// TIA Portal project "Alarms" (V15.1)

(* hardware
DEVICE "S71500/ET200MP station_1"  S7-1500 station
   slot 0: "Rail_0"  Rack  6ES7 590-1***0-0AA0
   slot 0: "PM 190W 120/230VAC"  PM 190W 120/230VAC  6EP1333-4BA00
   slot 1: "PLC_1"  CPU 1516-3 PN/DP  6ES7 516-3AN01-0AB0  V2.6
      slot 3: "CPU display_1"  6ES7591-1BA00-0AA0
   slot 2: "DQ 32x24VDC/0.5A HF_1"  DQ 32x24VDC/0.5A HF  6ES7 522-1BL01-0AB0  V1.1
   slot 3: "DI 32x24VDC HF_1"  DI 32x24VDC HF  6ES7 521-1BL00-0AB0  V2.1
   slot 4: "AQ 4xU/I ST_1"  AQ 4xU/I ST  6ES7 532-5HD00-0AB0  V2.2
   slot 5: "AI 8xU/I/RTD/TC ST_1"  AI 8xU/I/RTD/TC ST  6ES7 531-7KF00-0AB0  V2.2
DEVICE "HMI_1"  TP700 Comfort
   slot 0: "HMI_1"  TP700 Comfort  6AV2 124-0GC01-0AX0  15.1.0.0
   slot 1: "HMI_RT_1"  TP700 Comfort  6AV2 124-0GC01-0AX0  15.1.0.0
   slot 5: "HMI_1.IE_CP_1"  PROFINET Interface  15.0.1.0
      slot 1: "PROFINET Interface_1"  PROFINET Interface
         slot 1: "Port_1"  Port
         slot 2: "Port_2"  Port
   slot 7: "HMI_1.MPI/DP_CP_1"  MPI/DP Interface  15.0.1.0
*)

// ===== PLC "PLC_1"  CPU 1516-3 PN/DP =====

VAR_GLOBAL   // PLC tag table "Default tag table"
   "Clock_Byte" AT %MB0 : Byte;
   "Clock_10Hz" AT %M0.0 : Bool;
   "Clock_5Hz" AT %M0.1 : Bool;
   "Clock_2.5Hz" AT %M0.2 : Bool;
   "Clock_2Hz" AT %M0.3 : Bool;
   "Clock_1.25Hz" AT %M0.4 : Bool;
   "Clock_1Hz" AT %M0.5 : Bool;
   "Clock_0.625Hz" AT %M0.6 : Bool;
   "Clock_0.5Hz" AT %M0.7 : Bool;
   "System_Byte" AT %MB1 : Byte;
   "FirstScan" AT %M1.0 : Bool;
   "DiagStatusUpdate" AT %M1.1 : Bool;
   "AlwaysTRUE" AT %M1.2 : Bool;
   "AlwaysFALSE" AT %M1.3 : Bool;
   "System_Byte(1)" AT %MB1 : Byte;
   "System_Byte(2)" AT %MB1 : Byte;
END_VAR

VAR_GLOBAL   // PLC tag table "Full_Tag_Table"
   "Panel Emergency Stop" AT %I2.7 : Bool;
   "Start switch" AT %I0.2 : Bool;
   "Stop switch" AT %I0.3 : Bool;
   "Sort area IR" AT %I0.4 : Bool;
   "Sort Area Inductive" AT %I0.5 : Bool;
   "Sort Solenoid Sensor" AT %I0.6 : Bool;
   "Assembly Chute IR" AT %I0.7 : Bool;
   "Assembly Area Through Beam" AT %I1.1 : Bool;
   "Assembly Area Capacitor" AT %I1.2 : Bool;
   "Assembly Area Inductive" AT %I1.3 : Bool;
   "Reject Area IR" AT %I1.4 : Bool;
   "Reject Solenoid Sensor" AT %I1.5 : Bool;
   "Oven Through Beam" AT %I1.6 : Bool;
   "Loading Area Inductive" AT %I1.7 : Bool;
   "Chain Conveyor" AT %Q0.0 : Bool;
   "Sort Solenoid" AT %Q0.1 : Bool;
   "Reject Solenoid" AT %Q0.2 : Bool;
   "Rotary Solenoid" AT %Q0.3 : Bool;
   "Belt Conveyor Direction" AT %Q0.4 : Bool;
   "System Run_Green Lamp" AT %Q3.0 : Bool;
   "Sysyem Stop_Red Lamp" AT %Q3.2 : Bool;
   "Emergency stop" AT %I1.0 : Bool;
   "Ring Queue counter Full" AT %M4.0 : Bool;
   "Sort Solenoid error" AT %M4.3 : Bool;
   "Counter value" AT %MW0 : Int;
   "Reject Solenoid Error" AT %M4.7 : Bool;
   "HMI_Start" AT %M4.1 : Bool;
   "HMI_Stop" AT %M4.2 : Bool;
   "Counter Reset" AT %M4.4 : Bool;
   "Assembly Complete" AT %M4.5 : Bool;
   "Reset" AT %M4.6 : Bool;
   "HMI_Emergency_Stop" AT %M5.0 : Bool;
   "Ring Counter Value" AT %MW2 : Int;
   "Peg Counter Value" AT %MW6 : Int;
   "Assembly Counter Value" AT %MW8 : Int;
   "Connection_Successful" AT %M5.1 : Bool;
   "Connection_Disconnected" AT %M5.2 : Bool;
   "HMI_AssemDone" AT %M5.3 : Bool;
   "HMI_ConReset" AT %M5.4 : Bool;
   "HMI_SS_Alarm" AT %MW5 : Int;
   "Oven Temperature" AT %IW4 : Int;
   "Temperature control" AT %QW4 : Int;
   "Bipolar_SCALE" AT %M2000.0 : Bool;
   "Bipolar_UNSCALE" AT %M2000.1 : Bool;
   "Actual Retain Value" AT %MW100 : Word;
   "UNSCALE retain value" AT %MW15 : Word;
   "Real Temperature" AT %MD300 : Real;
   "Control value" AT %MW13 : Int;
   "ON/OFF Temperature" AT %MD9 : Real;
   "Temperature set point" AT %MD24 : Real;
   "ON/OFF Temperature set point" AT %MD20 : Real;
   "Save_Energy" AT %M28.0 : Bool;
   "Reset2" AT %M28.2 : Bool;
   "Em_Alarm" AT %M20.0 : Bool;
   "Alarm_Tag" AT %MW20 : Int;
   "PaEm_Alarm" AT %M20.1 : Bool;
   "SortSole_Alarm" AT %M20.2 : Bool;
   "RejectSole_Alarm" AT %M20.3 : Bool;
   "Count_Alarm" AT %M20.4 : Bool;
   "HMIReset" AT %M6.0 : Bool;
END_VAR

DATA_BLOCK "Automatic_Conveyor_DB"   // DB1
{ S7_Optimized_Access := 'TRUE' }
VERSION : 0.1
// stored: InstanceOfName Automatic_Conveyor
"Automatic_Conveyor"
BEGIN
END_DATA_BLOCK

DATA_BLOCK "Sort Solenoid Active_DB"   // DB2
{ S7_Optimized_Access := 'TRUE' }
VERSION : 0.1
// stored: InstanceOfName Sort Solenoid Active
"Sort Solenoid Active"
BEGIN
END_DATA_BLOCK

DATA_BLOCK "Solenoids Error_DB"   // DB3
{ S7_Optimized_Access := 'TRUE' }
VERSION : 0.1
// stored: InstanceOfName Solenoids Error
"Solenoids Error"
BEGIN
END_DATA_BLOCK

DATA_BLOCK "Rotary Solenoid Active_DB"   // DB4
{ S7_Optimized_Access := 'TRUE' }
VERSION : 0.1
// stored: InstanceOfName Rotary Solenoid Active
"Rotary Solenoid Active"
BEGIN
END_DATA_BLOCK

DATA_BLOCK "Counting_DB"   // DB5
{ S7_Optimized_Access := 'TRUE' }
VERSION : 0.1
// stored: InstanceOfName Counting
"Counting"
BEGIN
END_DATA_BLOCK

DATA_BLOCK "Solenoids Error_DB_1"   // DB6
{ S7_Optimized_Access := 'TRUE' }
VERSION : 0.1
// stored: InstanceOfName Solenoids Error
"Solenoids Error"
BEGIN
END_DATA_BLOCK

DATA_BLOCK "Component Queue Handling_DB"   // DB7
{ S7_Optimized_Access := 'TRUE' }
VERSION : 0.1
// stored: InstanceOfName Component Queue Handling
"Component Queue Handling"
BEGIN
END_DATA_BLOCK

DATA_BLOCK "Datablock"   // DB12
{ S7_Optimized_Access := 'TRUE' }
VERSION : 0.1
   VAR
      Sending_Data : Array[0..12] of Byte;
      Received_Data : Array[0..10] of Char;
      Send_Comm : Array[0..15] of Char;
   END_VAR
BEGIN
   Sending_Data[0] := 'A';
   Sending_Data[1] := 's';
   Sending_Data[2] := 's';
   Sending_Data[3] := 'e';
   Sending_Data[4] := 'm';
   Sending_Data[5] := 'b';
   Sending_Data[6] := 'l';
   Sending_Data[7] := 'y';
   Sending_Data[8] := ' ';
   Sending_Data[9] := 'D';
   Sending_Data[10] := 'o';
   Sending_Data[11] := 'n';
   Sending_Data[12] := 'e';
   Send_Comm[2] := 'o';
   Send_Comm[1] := 'r';
   Send_Comm[0] := 'P';
   Send_Comm[3] := 'c';
   Send_Comm[4] := 'e';
   Send_Comm[5] := 's';
   Send_Comm[6] := 's';
   Send_Comm[7] := ' ';
   Send_Comm[8] := 'S';
   Send_Comm[9] := 't';
   Send_Comm[10] := 'a';
   Send_Comm[11] := 'r';
   Send_Comm[12] := 't';
   Send_Comm[13] := 'e';
   Send_Comm[14] := 'd';
   Send_Comm[15] := '!';
END_DATA_BLOCK

DATA_BLOCK "TCP/IP Connection_DB"   // DB14
{ S7_Optimized_Access := 'TRUE' }
VERSION : 0.1
// stored: InstanceOfName TCP/IP Connection
"TCP/IP Connection"
BEGIN
END_DATA_BLOCK

DATA_BLOCK "Energy Saving_DB"   // DB17
{ S7_Optimized_Access := 'TRUE' }
VERSION : 0.1
// stored: InstanceOfName Energy Saving
"Energy Saving"
BEGIN
END_DATA_BLOCK

DATA_BLOCK "Alarm_DB"   // DB18
{ S7_Optimized_Access := 'TRUE' }
VERSION : 0.1
// stored: InstanceOfName Alarm
"Alarm"
BEGIN
END_DATA_BLOCK

// folder: System blocks/Program resources

DATA_BLOCK "PLC_1_Connection_DB"   // DB13
{ S7_Optimized_Access := 'TRUE' }
AUTHOR : SIMATIC
FAMILY : MC7Plus
NAME : TC_IP_v4
VERSION : 1.0
// stored: InstanceOfName TCON_IP_v4
"TCON_IP_v4"
BEGIN
   ID := 1;
   InterfaceId := 64;
   LocalPort := 2000;
   RemotePort := 10999;
   ActiveEstablished := true;
   RemoteAddress.ADDR[1] := 192;
   RemoteAddress.ADDR[2] := 168;
   RemoteAddress.ADDR[4] := 3;
END_DATA_BLOCK

// folder: (top level)

FUNCTION_BLOCK "Automatic_Conveyor"   // FB1, LAD
TITLE = Conveyors Automatic
{ S7_Optimized_Access := 'TRUE' }
VERSION : 0.1
   VAR_INPUT
      "Start Switch" : Bool;
      "Stop Switch" : Bool;
      "Emergency Stop" : Bool;
      "Panel Emergency Stop" : Bool;
      "Sort Solenoid Error" : Bool;
      "Reject Solenoid Error" : Bool;
      Reset : Bool;
      "Assembly Done" : Bool;
      H_Start : Bool;
      H_Stop : Bool;
      H_Emer_Stop : Bool;
      Save : Bool;
   END_VAR
   VAR_OUTPUT
      "System Enable_OK" : Bool;
      "System Enable_not_OK" : Bool;
      "Chain Conveyor" : Bool;
      "Belt Conveyor" : Bool;
   END_VAR
   VAR_IN_OUT
      Reset2 : Bool;
   END_VAR
   VAR
      Memory_Automatic_Start_Stop : Bool;
      Temp : Bool;
      SR_Temp : Bool;
      IEC_Timer_0_Instance_1 : TON_TIME;
      IEC_Timer_0_Instance_3 : TON_TIME;
   END_VAR
BEGIN

REGION Network 1: System Enable_OK and Conveyors run
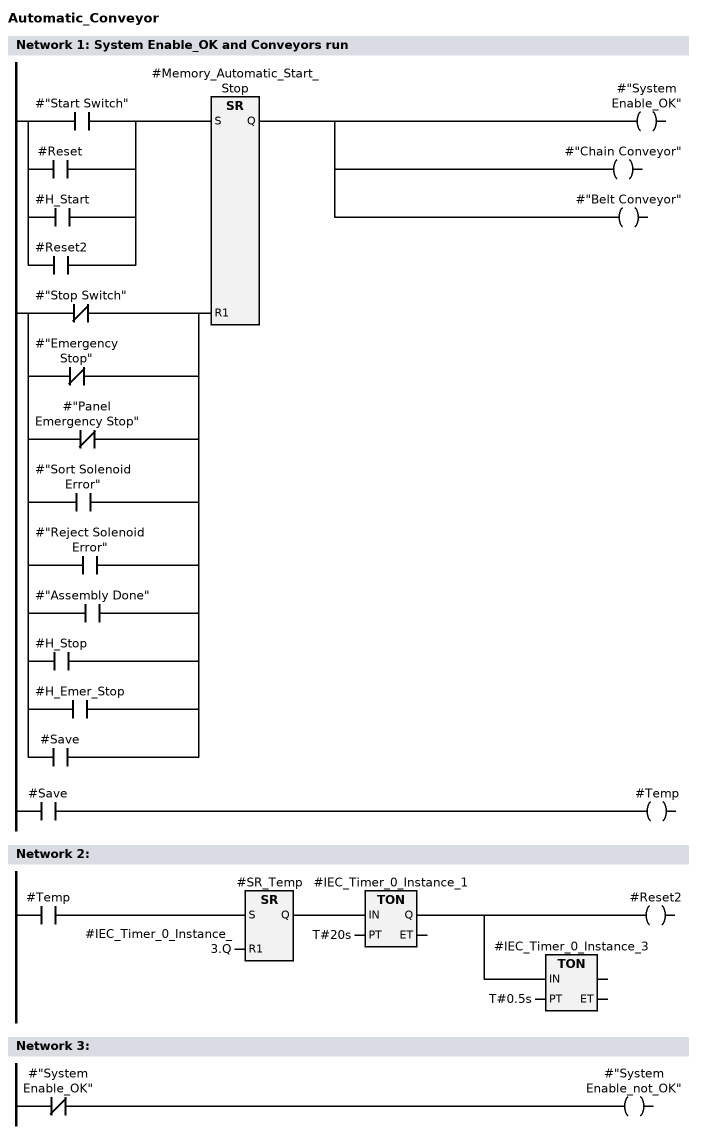
   RUNG wire#powerrail
      Contact( #"Start Switch" )
      wire#w1
      S_SR(operand := #Memory_Automatic_Start_Stop, r1 := wire#w2)
      wire#w3
      Coil( #"System Enable_OK" )
   END_RUNG
   RUNG wire#powerrail
      Contact( #Reset )
   END_RUNG wire#w1
   RUNG wire#powerrail
      Contact( #H_Start )
   END_RUNG wire#w1
   RUNG wire#powerrail
      Contact( #Reset2 )
   END_RUNG wire#w1
   RUNG wire#powerrail
      I_Contact( #"Stop Switch" )
   END_RUNG wire#w2
   RUNG wire#powerrail
      I_Contact( #"Emergency Stop" )
   END_RUNG wire#w2
   RUNG wire#powerrail
      I_Contact( #"Panel Emergency Stop" )
   END_RUNG wire#w2
   RUNG wire#powerrail
      Contact( #"Sort Solenoid Error" )
   END_RUNG wire#w2
   RUNG wire#powerrail
      Contact( #"Reject Solenoid Error" )
   END_RUNG wire#w2
   RUNG wire#powerrail
      Contact( #"Assembly Done" )
   END_RUNG wire#w2
   RUNG wire#powerrail
      Contact( #H_Stop )
   END_RUNG wire#w2
   RUNG wire#powerrail
      Contact( #H_Emer_Stop )
   END_RUNG wire#w2
   RUNG wire#powerrail
      Contact( #Save )
   END_RUNG wire#w2
   RUNG wire#w3
      Coil( #"Chain Conveyor" )
   END_RUNG
   RUNG wire#w3
      Coil( #"Belt Conveyor" )
   END_RUNG
   RUNG wire#powerrail
      Contact( #Save )
      Coil( #Temp )
   END_RUNG
   // the same network as SCL:
   IF #"Start Switch" OR #Reset OR #H_Start OR #Reset2 THEN
       #Memory_Automatic_Start_Stop := TRUE;   // SR flip-flop
   END_IF;
   IF NOT #"Stop Switch" OR NOT #"Emergency Stop" OR NOT #"Panel Emergency Stop" OR #"Sort Solenoid Error" OR #"Reject Solenoid Error" OR #"Assembly Done" OR #H_Stop OR #H_Emer_Stop OR #Save THEN
       #Memory_Automatic_Start_Stop := FALSE;
   END_IF;
   #"System Enable_OK" := #Memory_Automatic_Start_Stop;
   #"Chain Conveyor" := #Memory_Automatic_Start_Stop;
   #"Belt Conveyor" := #Memory_Automatic_Start_Stop;
   #Temp := #Save;
END_REGION

REGION Network 2
   IF #Temp THEN
       #SR_Temp := TRUE;   // SR flip-flop
   END_IF;
   IF #IEC_Timer_0_Instance_3.Q THEN #SR_Temp := FALSE; END_IF;
   #IEC_Timer_0_Instance_1(IN := #SR_Temp, PT := T#20s);   // TON
   #Reset2 := #IEC_Timer_0_Instance_1.Q;
   #IEC_Timer_0_Instance_3(IN := #IEC_Timer_0_Instance_1.Q, PT := T#0.5s);   // TON
END_REGION

REGION Network 3
   RUNG wire#powerrail
      I_Contact( #"System Enable_OK" )
      Coil( #"System Enable_not_OK" )
   END_RUNG
   // the same network as SCL:
   #"System Enable_not_OK" := NOT #"System Enable_OK";
END_REGION
END_FUNCTION_BLOCK

FUNCTION_BLOCK "Sort Solenoid Active"   // FB2, LAD
TITLE = Sort Solenoid Active
{ S7_Optimized_Access := 'TRUE' }
VERSION : 0.1
   VAR_INPUT
      "Sort Area IR" : Bool;
      "Sort Area Inductive" : Bool;
      "Ring Counter Full" : Bool;
   END_VAR
   VAR_OUTPUT
      "Sort Solenoid" : Bool;
   END_VAR
   VAR
      "Component Pass Delay" : Bool;
      "SR_Sort Solenoid on Timer" : Bool;
      "SR_Component Pass Delay" : Bool;
      IEC_Timer_0_Instance : TON_TIME;
      IEC_Timer_0_Instance_2 : TON_TIME;
   END_VAR
BEGIN

REGION Network 1: Sort Solenoid Active if Plastic Ring Present
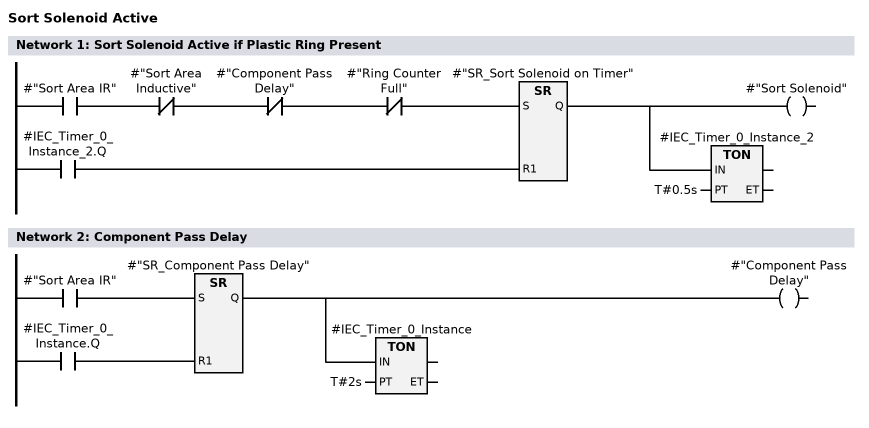
   IF #"Sort Area IR" AND NOT #"Sort Area Inductive" AND NOT #"Component Pass Delay" AND NOT #"Ring Counter Full" THEN
       #"SR_Sort Solenoid on Timer" := TRUE;   // SR flip-flop
   END_IF;
   IF #IEC_Timer_0_Instance_2.Q THEN #"SR_Sort Solenoid on Timer" := FALSE; END_IF;
   #"Sort Solenoid" := #"SR_Sort Solenoid on Timer";
   #IEC_Timer_0_Instance_2(IN := #"SR_Sort Solenoid on Timer", PT := T#0.5s);   // TON
END_REGION

REGION Network 2: Component Pass Delay
   IF #"Sort Area IR" THEN
       #"SR_Component Pass Delay" := TRUE;   // SR flip-flop
   END_IF;
   IF #IEC_Timer_0_Instance.Q THEN #"SR_Component Pass Delay" := FALSE; END_IF;
   #"Component Pass Delay" := #"SR_Component Pass Delay";
   #IEC_Timer_0_Instance(IN := #"SR_Component Pass Delay", PT := T#2s);   // TON
END_REGION
END_FUNCTION_BLOCK

FUNCTION_BLOCK "Solenoids Error"   // FB3, LAD
TITLE = Solenoid Error - Closed Loop Control
{ S7_Optimized_Access := 'TRUE' }
VERSION : 0.1
   VAR_INPUT
      "Solenoid on" : Bool;
      "Solenoid sensor" : Bool;
   END_VAR
   VAR_OUTPUT
      "Solenoid Error" : Bool;
   END_VAR
   VAR
      "Hold off delay" : Bool;
      IEC_Timer_0_Instance : TON_TIME;
   END_VAR
BEGIN

REGION Network 1: Solenoid Error
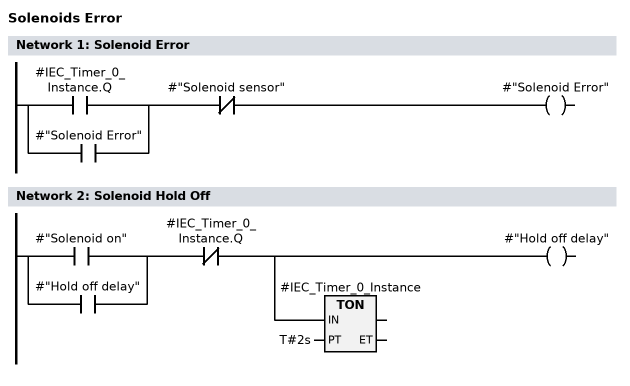
   RUNG wire#powerrail
      Contact( #IEC_Timer_0_Instance.Q )
      wire#w1
      I_Contact( #"Solenoid sensor" )
      Coil( #"Solenoid Error" )
   END_RUNG
   RUNG wire#powerrail
      Contact( #"Solenoid Error" )
   END_RUNG wire#w1
   // the same network as SCL:
   #"Solenoid Error" := (#IEC_Timer_0_Instance.Q OR #"Solenoid Error") AND NOT #"Solenoid sensor";
END_REGION

REGION Network 2: Solenoid Hold Off
   #"Hold off delay" := (#"Solenoid on" OR #"Hold off delay") AND NOT #IEC_Timer_0_Instance.Q;
   #IEC_Timer_0_Instance(IN := #"Hold off delay", PT := T#2s);   // TON
END_REGION
END_FUNCTION_BLOCK

FUNCTION_BLOCK "Counting"   // FB4, LAD
TITLE = Counting
{ S7_Optimized_Access := 'TRUE' }
VERSION : 0.1
// Incremental and Decremental counting
   VAR_INPUT
      "Sort Solenoid" : Bool;
      "Rotary Solenoid" : Bool;
      "Counter Reset" : Bool;
      "Sort Area Inductive" : Bool;
      "Sort Area IR" : Bool;
      "Assembly Complete" : Bool;
   END_VAR
   VAR_OUTPUT
      "Ring Queue counter full" : Bool;
      "Counter Value" : Int;
      "Ring CounterValue" : Int;
      "Peg CounterValue" : Int;
      "AssemblyCom CounterValue" : Int;
   END_VAR
   VAR RETAIN
      IEC_Counter_0_Instance : CTUD_INT;
      IEC_Counter_0_Instance_1 : CTU_INT;
      IEC_Counter_0_Instance_2 : CTU_INT;
      IEC_Counter_0_Instance_3 : CTU_INT;
   END_VAR
   VAR
      "Peg Count" : Bool;
      IEC_Timer_0_Instance : TOF_TIME;
   END_VAR
BEGIN

REGION Network 1: Counting
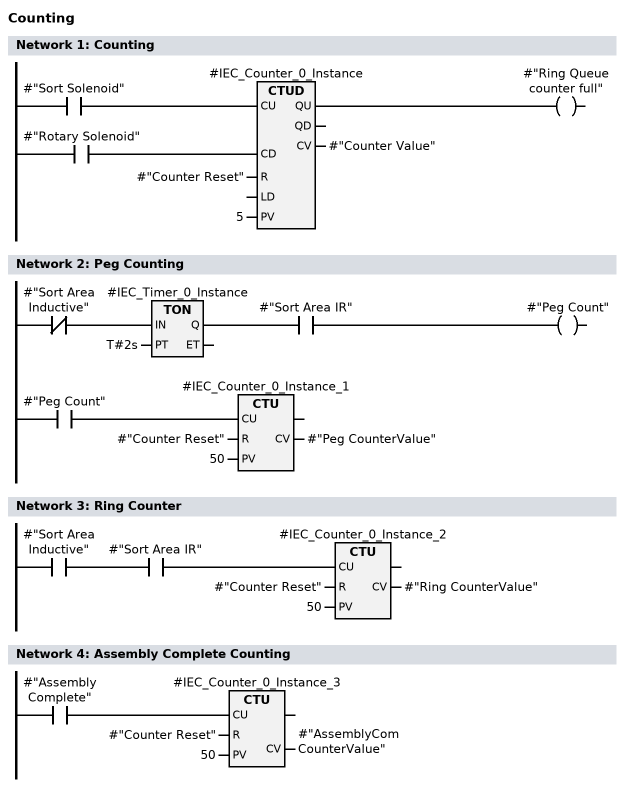
   #IEC_Counter_0_Instance(CU := #"Sort Solenoid",   // CTUD
                           CD := #"Rotary Solenoid",
                           R := #"Counter Reset",
                           PV := 5,
                           CV => #"Counter Value");
   #"Ring Queue counter full" := #IEC_Counter_0_Instance.QU;
END_REGION

REGION Network 2: Peg Counting
   #IEC_Timer_0_Instance(IN := NOT #"Sort Area Inductive", PT := T#2s);   // TON
   #"Peg Count" := #IEC_Timer_0_Instance.Q AND #"Sort Area IR";
   #IEC_Counter_0_Instance_1(CU := #"Peg Count", R := #"Counter Reset", PV := 50, CV => #"Peg CounterValue");   // CTU
END_REGION

REGION Network 3: Ring Counter
   #IEC_Counter_0_Instance_2(CU := #"Sort Area Inductive" AND #"Sort Area IR",   // CTU
                           R := #"Counter Reset",
                           PV := 50,
                           CV => #"Ring CounterValue");
END_REGION

REGION Network 4: Assembly Complete Counting
   #IEC_Counter_0_Instance_3(CU := #"Assembly Complete",   // CTU
                           R := #"Counter Reset",
                           PV := 50,
                           CV => #"AssemblyCom CounterValue");
END_REGION
END_FUNCTION_BLOCK

FUNCTION_BLOCK "Rotary Solenoid Active"   // FB5, LAD
TITLE = Rotary Solenoid Active
{ S7_Optimized_Access := 'TRUE' }
VERSION : 0.1
   VAR_INPUT
      "Rotary Area IR" : Bool;
   END_VAR
   VAR_OUTPUT
      "Rotary Solenoid" : Bool;
   END_VAR
   VAR
      "SR_Component Pass Delay" : Bool;
      "Component Pass Delay" : Bool;
      IEC_Timer_0_Instance : TON_TIME;
      IEC_Timer_0_Instance_2 : TON_TIME;
      "SR Rotary Solenoid on Timer" : Bool;
      IEC_Timer_0_Instance_1 : TON_TIME;
   END_VAR
BEGIN

REGION Network 1: Rotary Solenoid Activation
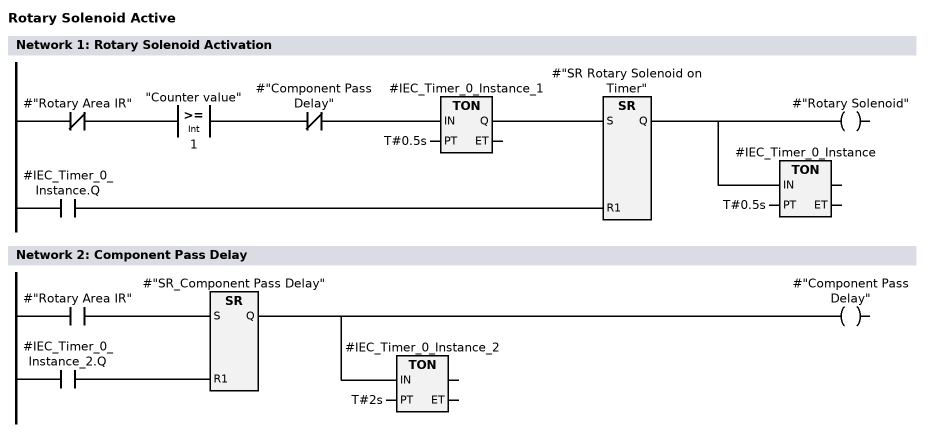
   #IEC_Timer_0_Instance_1(IN := NOT #"Rotary Area IR" AND ("Counter value" >= 1) AND NOT #"Component Pass Delay",   // TON
                           PT := T#0.5s);
   IF #IEC_Timer_0_Instance_1.Q THEN
       #"SR Rotary Solenoid on Timer" := TRUE;   // SR flip-flop
   END_IF;
   IF #IEC_Timer_0_Instance.Q THEN #"SR Rotary Solenoid on Timer" := FALSE; END_IF;
   #"Rotary Solenoid" := #"SR Rotary Solenoid on Timer";
   #IEC_Timer_0_Instance(IN := #"SR Rotary Solenoid on Timer", PT := T#0.5s);   // TON
END_REGION

REGION Network 2: Component Pass Delay
   IF #"Rotary Area IR" THEN
       #"SR_Component Pass Delay" := TRUE;   // SR flip-flop
   END_IF;
   IF #IEC_Timer_0_Instance_2.Q THEN #"SR_Component Pass Delay" := FALSE; END_IF;
   #"Component Pass Delay" := #"SR_Component Pass Delay";
   #IEC_Timer_0_Instance_2(IN := #"SR_Component Pass Delay", PT := T#2s);   // TON
END_REGION
END_FUNCTION_BLOCK

FUNCTION_BLOCK "Component Queue Handling"   // FB6, LAD
TITLE = Component Queue Handling
{ S7_Optimized_Access := 'TRUE' }
VERSION : 0.1
   VAR_INPUT
      "Start Switch" : Bool;
      "Assembly Area Capacitive" : Bool;
      "Assembly Area Inductive" : Bool;
      "Reject Area IR" : Bool;
      "Assembly Area Through Beam" : Bool;
   END_VAR
   VAR_OUTPUT
      "Reject Solenoid" : Bool;
      "Assembly Done" : Bool;
      HMIReset : Bool;
      HMI_AssDone : Bool;
   END_VAR
   VAR
      "Pointer Register" : Word;
      "Data Register" : Word;
      "SHL Memory" : Bool;
      "SHR Memory" : Bool;
      "And Result" : Word;
      SR_Reject : Bool;
      IEC_Timer_0_Instance : TON_TIME;
      "Assembly Complete" : Bool;
      IEC_Timer_0_Instance_1 : TON_TIME;
      "SR_Assembly Done" : Bool;
      IEC_Timer_0_Instance_2 : TON_TIME;
      SR_Stop : Bool;
      IEC_Timer_0_Instance_5 : TON_TIME;
      SR_Inductive : Bool;
      IEC_Timer_0_Instance_6 : TON_TIME;
      IEC_Timer_0_Instance_7 : TON_TIME;
      IEC_Timer_0_Instance_8 : TON_TIME;
      HMI_SR : Bool;
      IEC_Timer_0_Instance_3 : TON_TIME;
   END_VAR
   VAR_TEMP   // added for the SCL form of the ladder/FBD networks
      _w1 : Bool;
   END_VAR
BEGIN

REGION Network 1: Data and pointer register
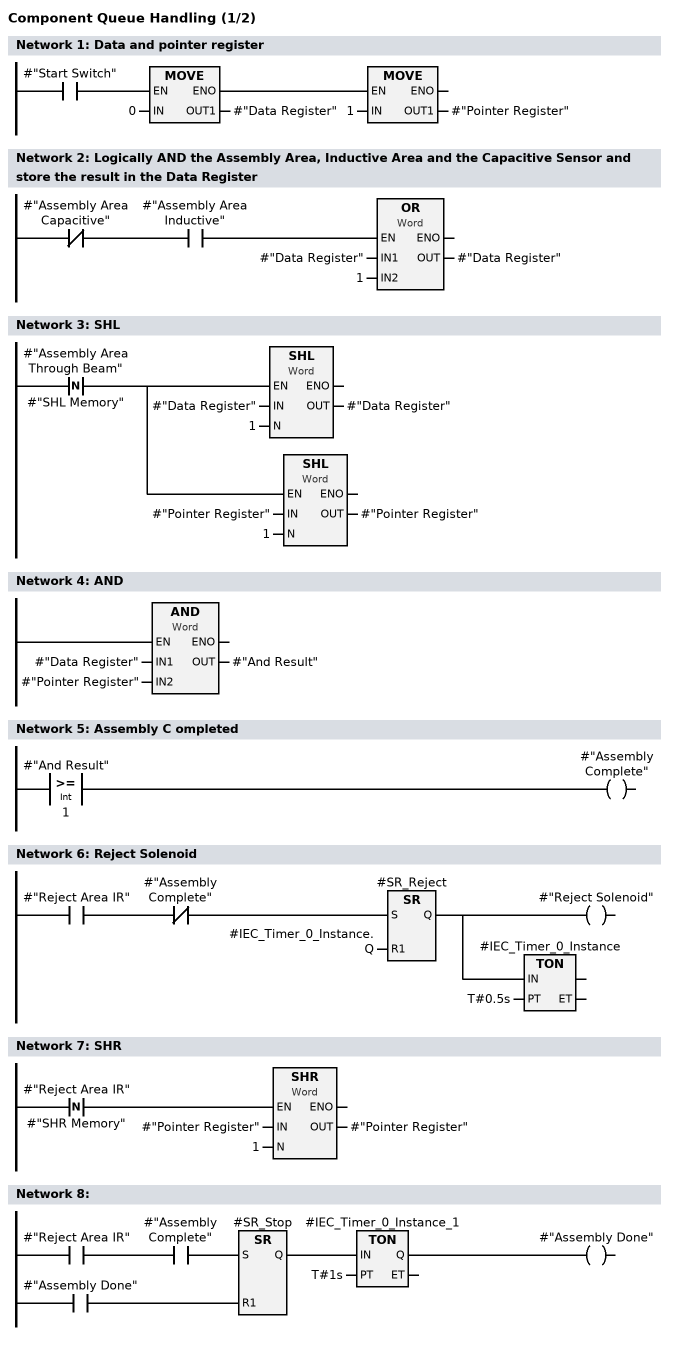
   RUNG wire#powerrail
      Contact( #"Start Switch" )
      Move(in := 0, out1 => #"Data Register")
      Move(in := 1, out1 => #"Pointer Register")
   END_RUNG
   // the same network as SCL:
   IF #"Start Switch" THEN
       #"Data Register" := 0;
       #"Pointer Register" := 1;
   END_IF;
END_REGION

REGION Network 2: Logically AND the Assembly Area, Inductive Area and the Capacitive Sensor and store the result in the Data Register
   IF NOT #"Assembly Area Capacitive" AND #"Assembly Area Inductive" THEN
       #"Data Register" := #"Data Register" OR 1;
   END_IF;
END_REGION

REGION Network 3: SHL
   RUNG wire#powerrail
      N_Contact(operand := #"Assembly Area Through Beam", bit := #"SHL Memory")
      wire#w1
      { S7_Templates := "SrcType := Word" } Shl(in := #"Data Register", n := 1, out => #"Data Register")
   END_RUNG
   RUNG wire#w1
      { S7_Templates := "SrcType := Word" } Shl(in := #"Pointer Register", n := 1, out => #"Pointer Register")
   END_RUNG
   // the same network as SCL:
   #_w1 := NOT #"Assembly Area Through Beam" AND #"SHL Memory";   // falling edge of #"Assembly Area Through Beam"
   #"SHL Memory" := #"Assembly Area Through Beam";
   IF #_w1 THEN
       #"Data Register" := SHL(IN := #"Data Register", N := 1);
       #"Pointer Register" := SHL(IN := #"Pointer Register", N := 1);
   END_IF;
END_REGION

REGION Network 4: AND
   RUNG wire#powerrail
      { S7_Templates := "SrcType := Word" } And(in1 := #"Data Register", in2 := #"Pointer Register", out => #"And Result")
   END_RUNG
   // the same network as SCL:
   #"And Result" := #"Data Register" AND #"Pointer Register";
END_REGION

REGION Network 5: Assembly C ompleted
   RUNG wire#powerrail
      { S7_Templates := "SrcType := Int" } GE_Contact(in1 := #"And Result", in2 := 1)
      Coil( #"Assembly Complete" )
   END_RUNG
   // the same network as SCL:
   #"Assembly Complete" := #"And Result" >= 1;
END_REGION

REGION Network 6: Reject Solenoid
   IF #"Reject Area IR" AND NOT #"Assembly Complete" THEN
       #SR_Reject := TRUE;   // SR flip-flop
   END_IF;
   IF #IEC_Timer_0_Instance.Q THEN #SR_Reject := FALSE; END_IF;
   #"Reject Solenoid" := #SR_Reject;
   #IEC_Timer_0_Instance(IN := #SR_Reject, PT := T#0.5s);   // TON
END_REGION

REGION Network 7: SHR
   RUNG wire#powerrail
      N_Contact(operand := #"Reject Area IR", bit := #"SHR Memory")
      { S7_Templates := "SrcType := Word" } Shr(in := #"Pointer Register", n := 1, out => #"Pointer Register")
   END_RUNG
   // the same network as SCL:
   #_w1 := NOT #"Reject Area IR" AND #"SHR Memory";   // falling edge of #"Reject Area IR"
   #"SHR Memory" := #"Reject Area IR";
   IF #_w1 THEN #"Pointer Register" := SHR(IN := #"Pointer Register", N := 1); END_IF;
END_REGION

REGION Network 8
   IF #"Reject Area IR" AND #"Assembly Complete" THEN
       #SR_Stop := TRUE;   // SR flip-flop
   END_IF;
   IF #"Assembly Done" THEN #SR_Stop := FALSE; END_IF;
   #IEC_Timer_0_Instance_1(IN := #SR_Stop, PT := T#1s);   // TON
   #"Assembly Done" := #IEC_Timer_0_Instance_1.Q;
END_REGION

REGION Network 9
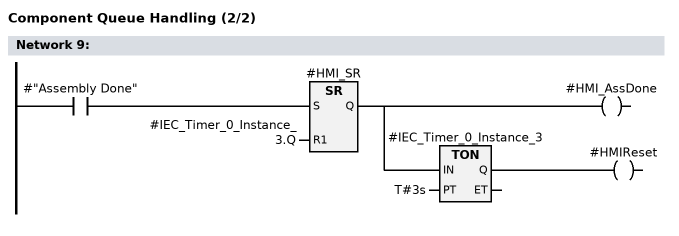
   IF #"Assembly Done" THEN
       #HMI_SR := TRUE;   // SR flip-flop
   END_IF;
   IF #IEC_Timer_0_Instance_3.Q THEN #HMI_SR := FALSE; END_IF;
   #HMI_AssDone := #HMI_SR;
   #IEC_Timer_0_Instance_3(IN := #HMI_SR, PT := T#3s);   // TON
   #HMIReset := #IEC_Timer_0_Instance_3.Q;
END_REGION
END_FUNCTION_BLOCK

FUNCTION_BLOCK "TCP/IP Connection"   // FB7, LAD
TITLE = Connection
{ S7_Optimized_Access := 'TRUE' }
VERSION : 0.1
// TCP/IP Connection
   VAR_OUTPUT
      "Connection Successful" : Bool;
      "Connection Disconnected" : Bool;
   END_VAR
   VAR
      TCON : Struct
         DONE : Bool;
         BUSY : Bool;
         ERROR : Bool;
         STATUS : UInt;
         DONESAVE : Bool;
      END_STRUCT;
      TDISCON : Struct
         DONE : Bool;
         REQ : Bool;
         BUSY : Bool;
         ERROR : Bool;
         STATUS : UInt;
      END_STRUCT;
      TSEND : Struct
         REQ : Bool;
         DONE : Bool;
         BUSY : Bool;
         ERROR : Bool;
         STATUS : UInt;
      END_STRUCT;
      TRCV : Struct
         EN_R : Bool;
         NDR : Bool;
         BUSY : Bool;
         ERROR : Bool;
         STATUS : UInt;
         RCVD_LEN : UInt;
      END_STRUCT;
      TSEND_Comm : Struct
         REQ : Bool;
         DONE : Bool;
         BUSY : Bool;
         ERROR : Bool;
         STATUS : UInt;
      END_STRUCT;
      "Received String" : String;
      IEC_Timer_0_Instance : TON_TIME;
      SR_Connection : Bool;
      SR_Disconnect : Bool;
      IEC_Timer_0_Instance_1 : TON_TIME;
   END_VAR
BEGIN

REGION Network 1: TCON
   // Establish connection between PLC and Laptop
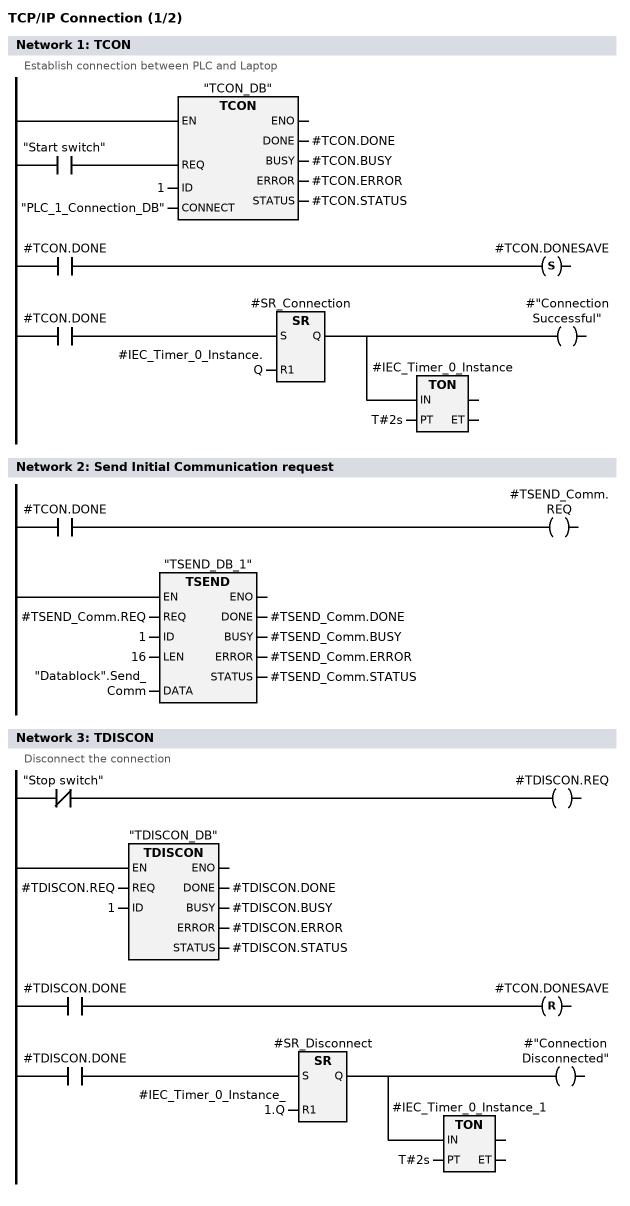
   "TCON_DB"(REQ := "Start switch",   // TCON
             ID := 1,
             CONNECT := "PLC_1_Connection_DB",
             DONE => #TCON.DONE,
             BUSY => #TCON.BUSY,
             ERROR => #TCON.ERROR,
             STATUS => #TCON.STATUS);
   IF #TCON.DONE THEN
       #TCON.DONESAVE := TRUE;
       #SR_Connection := TRUE;   // SR flip-flop
   END_IF;
   IF #IEC_Timer_0_Instance.Q THEN #SR_Connection := FALSE; END_IF;
   #"Connection Successful" := #SR_Connection;
   #IEC_Timer_0_Instance(IN := #SR_Connection, PT := T#2s);   // TON
END_REGION

REGION Network 2: Send Initial Communication request
   #TSEND_Comm.REQ := #TCON.DONE;
   "TSEND_DB_1"(REQ := #TSEND_Comm.REQ,   // TSEND
                ID := 1,
                LEN := 16,
                DATA := "Datablock".Send_Comm,
                DONE => #TSEND_Comm.DONE,
                BUSY => #TSEND_Comm.BUSY,
                ERROR => #TSEND_Comm.ERROR,
                STATUS => #TSEND_Comm.STATUS);
END_REGION

REGION Network 3: TDISCON
   // Disconnect the connection
   #TDISCON.REQ := NOT "Stop switch";
   "TDISCON_DB"(REQ := #TDISCON.REQ,   // TDISCON
                ID := 1,
                DONE => #TDISCON.DONE,
                BUSY => #TDISCON.BUSY,
                ERROR => #TDISCON.ERROR,
                STATUS => #TDISCON.STATUS);
   IF #TDISCON.DONE THEN
       #TCON.DONESAVE := FALSE;
       #SR_Disconnect := TRUE;   // SR flip-flop
   END_IF;
   IF #IEC_Timer_0_Instance_1.Q THEN #SR_Disconnect := FALSE; END_IF;
   #"Connection Disconnected" := #SR_Disconnect;
   #IEC_Timer_0_Instance_1(IN := #SR_Disconnect, PT := T#2s);   // TON
END_REGION

REGION Network 4: TSEND
   // Send Data
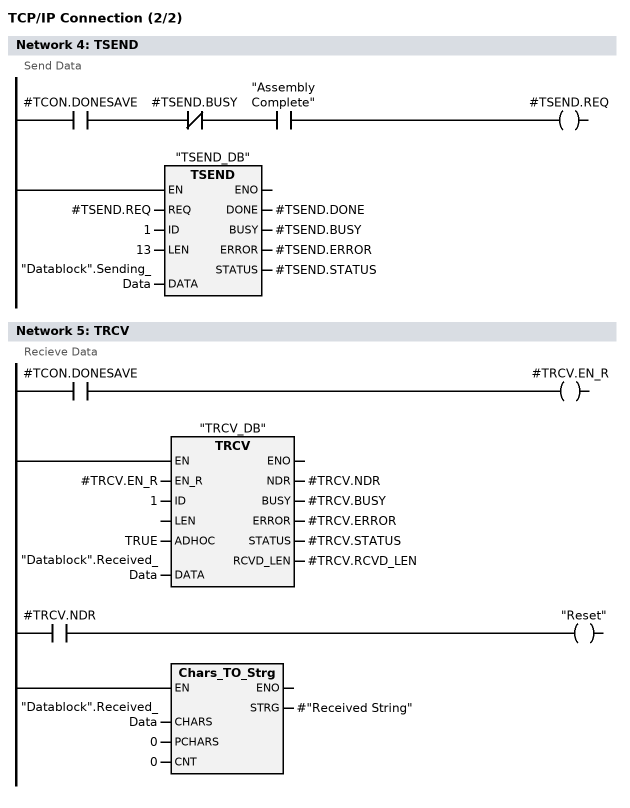
   #TSEND.REQ := #TCON.DONESAVE AND NOT #TSEND.BUSY AND "Assembly Complete";
   "TSEND_DB"(REQ := #TSEND.REQ,   // TSEND
              ID := 1,
              LEN := 13,
              DATA := "Datablock".Sending_Data,
              DONE => #TSEND.DONE,
              BUSY => #TSEND.BUSY,
              ERROR => #TSEND.ERROR,
              STATUS => #TSEND.STATUS);
END_REGION

REGION Network 5: TRCV
   // Recieve Data
   // no SCL statement known for Chars_TO_Strg: written as a call
   #TRCV.EN_R := #TCON.DONESAVE;
   "TRCV_DB"(EN_R := #TRCV.EN_R,   // TRCV
             ID := 1,
             ADHOC := TRUE,
             DATA := "Datablock".Received_Data,
             NDR => #TRCV.NDR,
             BUSY => #TRCV.BUSY,
             ERROR => #TRCV.ERROR,
             STATUS => #TRCV.STATUS,
             RCVD_LEN => #TRCV.RCVD_LEN);
   "Reset" := #TRCV.NDR;
   Chars_TO_Strg(Chars := "Datablock".Received_Data, pChars := 0, Cnt := 0, Strg => #"Received String");
END_REGION
END_FUNCTION_BLOCK

FUNCTION_BLOCK "Energy Saving"   // FB8, LAD
TITLE = Energy Saving
{ S7_Optimized_Access := 'TRUE' }
VERSION : 0.1
   VAR_INPUT
      "Start Switch" : Bool;
      "Sort IR sensor" : Bool;
      "System Enable Ok" : Bool;
   END_VAR
   VAR_OUTPUT
      Save : Bool;
   END_VAR
   VAR
      SR_Start : Bool;
      IEC_Timer_0_Instance : TON_TIME;
      IEC_Timer_0_Instance_3 : TON_TIME;
      SR_IR : Bool;
      IEC_Timer_0_Instance_1 : TON_TIME;
   END_VAR
BEGIN

REGION Network 1: Stop the belt if no peg/ring is present on the belt for 1min, reset after 20sec and the process repeats.
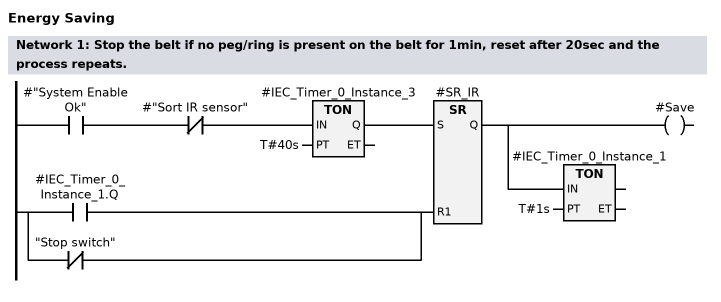
   #IEC_Timer_0_Instance_3(IN := #"System Enable Ok" AND NOT #"Sort IR sensor", PT := T#40s);   // TON
   IF #IEC_Timer_0_Instance_3.Q THEN
       #SR_IR := TRUE;   // SR flip-flop
   END_IF;
   IF #IEC_Timer_0_Instance_1.Q OR NOT "Stop switch" THEN #SR_IR := FALSE; END_IF;
   #Save := #SR_IR;
   #IEC_Timer_0_Instance_1(IN := #SR_IR, PT := T#1s);   // TON
END_REGION
END_FUNCTION_BLOCK

FUNCTION_BLOCK "Alarm"   // FB9, LAD
TITLE = Alarms
{ S7_Optimized_Access := 'TRUE' }
VERSION : 0.1
BEGIN

REGION Network 1
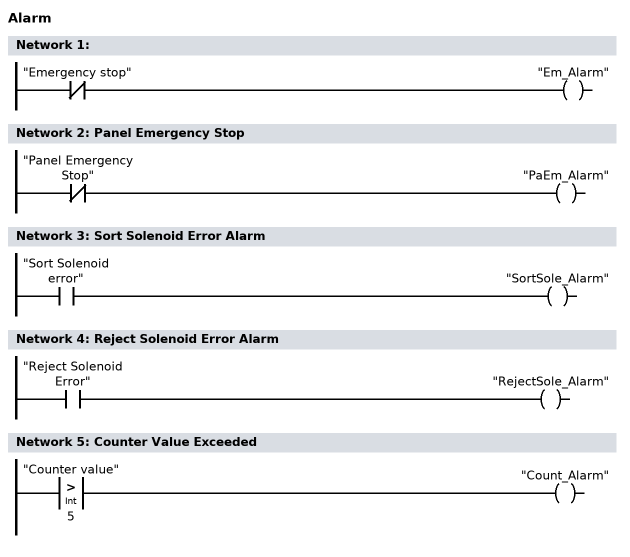
   RUNG wire#powerrail
      I_Contact( "Emergency stop" )
      Coil( "Em_Alarm" )
   END_RUNG
   // the same network as SCL:
   "Em_Alarm" := NOT "Emergency stop";
END_REGION

REGION Network 2: Panel Emergency Stop
   RUNG wire#powerrail
      I_Contact( "Panel Emergency Stop" )
      Coil( "PaEm_Alarm" )
   END_RUNG
   // the same network as SCL:
   "PaEm_Alarm" := NOT "Panel Emergency Stop";
END_REGION

REGION Network 3: Sort Solenoid Error Alarm
   RUNG wire#powerrail
      Contact( "Sort Solenoid error" )
      Coil( "SortSole_Alarm" )
   END_RUNG
   // the same network as SCL:
   "SortSole_Alarm" := "Sort Solenoid error";
END_REGION

REGION Network 4: Reject Solenoid Error Alarm
   RUNG wire#powerrail
      Contact( "Reject Solenoid Error" )
      Coil( "RejectSole_Alarm" )
   END_RUNG
   // the same network as SCL:
   "RejectSole_Alarm" := "Reject Solenoid Error";
END_REGION

REGION Network 5: Counter Value Exceeded
   RUNG wire#powerrail
      { S7_Templates := "SrcType := Int" } GT_Contact(in1 := "Counter value", in2 := 5)
      Coil( "Count_Alarm" )
   END_RUNG
   // the same network as SCL:
   "Count_Alarm" := "Counter value" > 5;
END_REGION
END_FUNCTION_BLOCK

FUNCTION "SCALE" : Void   // FC1, LAD
{ S7_Optimized_Access := 'TRUE' }
VERSION : 0.1
   VAR_INPUT
      "Input Analog Signal" : Int;
      "High Limit" : Real;
      "Low Limit" : Real;
      Bipolar : Bool;
   END_VAR
   VAR_OUTPUT
      "Real Physical Value" : Real;
      "Retain Value" : Word;
   END_VAR
BEGIN

REGION Network 1
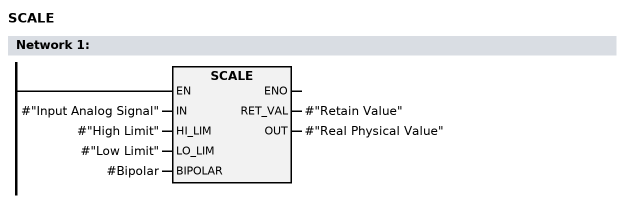
   #"Retain Value" := SCALE(IN := #"Input Analog Signal",
                           HI_LIM := #"High Limit",
                           LO_LIM := #"Low Limit",
                           BIPOLAR := #Bipolar,
                           OUT => #"Real Physical Value");
END_REGION
END_FUNCTION

FUNCTION "UNSCALE" : Void   // FC2, LAD
{ S7_Optimized_Access := 'TRUE' }
VERSION : 0.1
   VAR_INPUT
      "Input to unscale" : Real;
      "High Limit" : Real;
      "Low Limit" : Real;
      Bipolar : Bool;
   END_VAR
   VAR_OUTPUT
      "Output Analog Signal" : Int;
      "Retain Value" : Word;
   END_VAR
BEGIN

REGION Network 1: Unscale
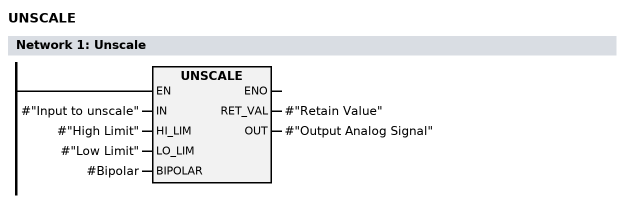
   #"Retain Value" := UNSCALE(IN := #"Input to unscale",
                           HI_LIM := #"High Limit",
                           LO_LIM := #"Low Limit",
                           BIPOLAR := #Bipolar,
                           OUT => #"Output Analog Signal");
END_REGION
END_FUNCTION

ORGANIZATION_BLOCK "Main"   // OB1, LAD, ProgramCycle
TITLE = "Main Program Sweep (Cycle)"
{ S7_Optimized_Access := 'TRUE' }
VERSION : 0.1
   VAR_INPUT
      Initial_Call : Bool;   // Initial call of this OB
      Remanence : Bool;   // =True, if remanent data are available
   END_VAR
BEGIN

REGION Network 1: System run ok and conveyors start
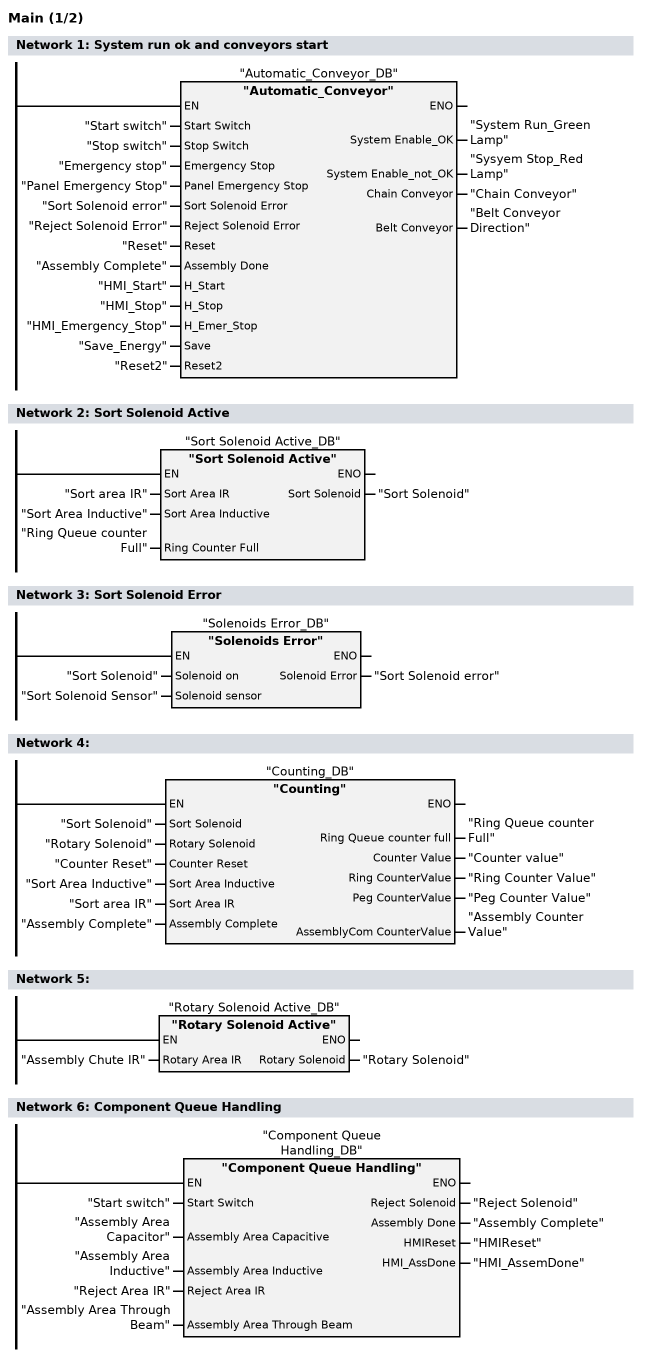
   RUNG wire#powerrail
      "Automatic_Conveyor_DB"("Start Switch" := "Start switch", "Stop Switch" := "Stop switch", "Emergency Stop" := "Emergency stop", "Panel Emergency Stop" := "Panel Emergency Stop", "Sort Solenoid Error" := "Sort Solenoid error", "Reject Solenoid Error" := "Reject Solenoid Error", Reset := "Reset", "Assembly Done" := "Assembly Complete", H_Start := "HMI_Start", H_Stop := "HMI_Stop", H_Emer_Stop := "HMI_Emergency_Stop", Save := "Save_Energy", Reset2 := "Reset2", "System Enable_OK" => "System Run_Green Lamp", "System Enable_not_OK" => "Sysyem Stop_Red Lamp", "Chain Conveyor" => "Chain Conveyor", "Belt Conveyor" => "Belt Conveyor Direction")
   END_RUNG
   // the same network as SCL:
   "Automatic_Conveyor_DB"("Start Switch" := "Start switch",   // "Automatic_Conveyor"
                           "Stop Switch" := "Stop switch",
                           "Emergency Stop" := "Emergency stop",
                           "Panel Emergency Stop" := "Panel Emergency Stop",
                           "Sort Solenoid Error" := "Sort Solenoid error",
                           "Reject Solenoid Error" := "Reject Solenoid Error",
                           Reset := "Reset",
                           "Assembly Done" := "Assembly Complete",
                           H_Start := "HMI_Start",
                           H_Stop := "HMI_Stop",
                           H_Emer_Stop := "HMI_Emergency_Stop",
                           Save := "Save_Energy",
                           Reset2 := "Reset2",
                           "System Enable_OK" => "System Run_Green Lamp",
                           "System Enable_not_OK" => "Sysyem Stop_Red Lamp",
                           "Chain Conveyor" => "Chain Conveyor",
                           "Belt Conveyor" => "Belt Conveyor Direction");
END_REGION

REGION Network 2: Sort Solenoid Active
   RUNG wire#powerrail
      "Sort Solenoid Active_DB"("Sort Area IR" := "Sort area IR", "Sort Area Inductive" := "Sort Area Inductive", "Ring Counter Full" := "Ring Queue counter Full", "Sort Solenoid" => "Sort Solenoid")
   END_RUNG
   // the same network as SCL:
   "Sort Solenoid Active_DB"("Sort Area IR" := "Sort area IR",   // "Sort Solenoid Active"
                           "Sort Area Inductive" := "Sort Area Inductive",
                           "Ring Counter Full" := "Ring Queue counter Full",
                           "Sort Solenoid" => "Sort Solenoid");
END_REGION

REGION Network 3: Sort Solenoid Error
   RUNG wire#powerrail
      "Solenoids Error_DB"("Solenoid on" := "Sort Solenoid", "Solenoid sensor" := "Sort Solenoid Sensor", "Solenoid Error" => "Sort Solenoid error")
   END_RUNG
   // the same network as SCL:
   "Solenoids Error_DB"("Solenoid on" := "Sort Solenoid",   // "Solenoids Error"
                        "Solenoid sensor" := "Sort Solenoid Sensor",
                        "Solenoid Error" => "Sort Solenoid error");
END_REGION

REGION Network 4
   RUNG wire#powerrail
      "Counting_DB"("Sort Solenoid" := "Sort Solenoid", "Rotary Solenoid" := "Rotary Solenoid", "Counter Reset" := "Counter Reset", "Sort Area Inductive" := "Sort Area Inductive", "Sort Area IR" := "Sort area IR", "Assembly Complete" := "Assembly Complete", "Ring Queue counter full" => "Ring Queue counter Full", "Counter Value" => "Counter value", "Ring CounterValue" => "Ring Counter Value", "Peg CounterValue" => "Peg Counter Value", "AssemblyCom CounterValue" => "Assembly Counter Value")
   END_RUNG
   // the same network as SCL:
   "Counting_DB"("Sort Solenoid" := "Sort Solenoid",   // "Counting"
                 "Rotary Solenoid" := "Rotary Solenoid",
                 "Counter Reset" := "Counter Reset",
                 "Sort Area Inductive" := "Sort Area Inductive",
                 "Sort Area IR" := "Sort area IR",
                 "Assembly Complete" := "Assembly Complete",
                 "Ring Queue counter full" => "Ring Queue counter Full",
                 "Counter Value" => "Counter value",
                 "Ring CounterValue" => "Ring Counter Value",
                 "Peg CounterValue" => "Peg Counter Value",
                 "AssemblyCom CounterValue" => "Assembly Counter Value");
END_REGION

REGION Network 5
   RUNG wire#powerrail
      "Rotary Solenoid Active_DB"("Rotary Area IR" := "Assembly Chute IR", "Rotary Solenoid" => "Rotary Solenoid")
   END_RUNG
   // the same network as SCL:
   "Rotary Solenoid Active_DB"("Rotary Area IR" := "Assembly Chute IR", "Rotary Solenoid" => "Rotary Solenoid");   // "Rotary Solenoid Active"
END_REGION

REGION Network 6: Component Queue Handling
   RUNG wire#powerrail
      "Component Queue Handling_DB"("Start Switch" := "Start switch", "Assembly Area Capacitive" := "Assembly Area Capacitor", "Assembly Area Inductive" := "Assembly Area Inductive", "Reject Area IR" := "Reject Area IR", "Assembly Area Through Beam" := "Assembly Area Through Beam", "Reject Solenoid" => "Reject Solenoid", "Assembly Done" => "Assembly Complete", HMIReset => "HMIReset", HMI_AssDone => "HMI_AssemDone")
   END_RUNG
   // the same network as SCL:
   "Component Queue Handling_DB"("Start Switch" := "Start switch",   // "Component Queue Handling"
                           "Assembly Area Capacitive" := "Assembly Area Capacitor",
                           "Assembly Area Inductive" := "Assembly Area Inductive",
                           "Reject Area IR" := "Reject Area IR",
                           "Assembly Area Through Beam" := "Assembly Area Through Beam",
                           "Reject Solenoid" => "Reject Solenoid",
                           "Assembly Done" => "Assembly Complete",
                           HMIReset => "HMIReset",
                           HMI_AssDone => "HMI_AssemDone");
END_REGION

REGION Network 7: Reject Area Solenoid Error
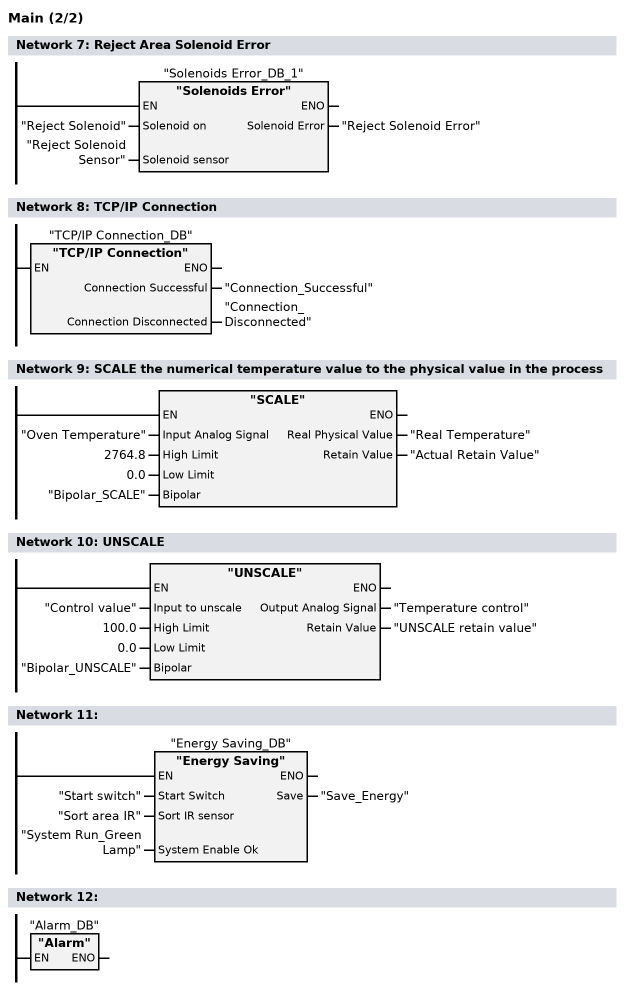
   RUNG wire#powerrail
      "Solenoids Error_DB_1"("Solenoid on" := "Reject Solenoid", "Solenoid sensor" := "Reject Solenoid Sensor", "Solenoid Error" => "Reject Solenoid Error")
   END_RUNG
   // the same network as SCL:
   "Solenoids Error_DB_1"("Solenoid on" := "Reject Solenoid",   // "Solenoids Error"
                          "Solenoid sensor" := "Reject Solenoid Sensor",
                          "Solenoid Error" => "Reject Solenoid Error");
END_REGION

REGION Network 8: TCP/IP Connection
   RUNG wire#powerrail
      "TCP/IP Connection_DB"("Connection Successful" => "Connection_Successful", "Connection Disconnected" => "Connection_Disconnected")
   END_RUNG
   // the same network as SCL:
   "TCP/IP Connection_DB"("Connection Successful" => "Connection_Successful",   // "TCP/IP Connection"
                          "Connection Disconnected" => "Connection_Disconnected");
END_REGION

REGION Network 9: SCALE the numerical temperature value to the physical value in the process
   RUNG wire#powerrail
      "SCALE"("Input Analog Signal" := "Oven Temperature", "High Limit" := 2764.8, "Low Limit" := 0.0, Bipolar := "Bipolar_SCALE", "Real Physical Value" => "Real Temperature", "Retain Value" => "Actual Retain Value")
   END_RUNG
   // the same network as SCL:
   "SCALE"("Input Analog Signal" := "Oven Temperature",
           "High Limit" := 2764.8,
           "Low Limit" := 0.0,
           Bipolar := "Bipolar_SCALE",
           "Real Physical Value" => "Real Temperature",
           "Retain Value" => "Actual Retain Value");
END_REGION

REGION Network 10: UNSCALE
   RUNG wire#powerrail
      "UNSCALE"("Input to unscale" := "Control value", "High Limit" := 100.0, "Low Limit" := 0.0, Bipolar := "Bipolar_UNSCALE", "Output Analog Signal" => "Temperature control", "Retain Value" => "UNSCALE retain value")
   END_RUNG
   // the same network as SCL:
   "UNSCALE"("Input to unscale" := "Control value",
             "High Limit" := 100.0,
             "Low Limit" := 0.0,
             Bipolar := "Bipolar_UNSCALE",
             "Output Analog Signal" => "Temperature control",
             "Retain Value" => "UNSCALE retain value");
END_REGION

REGION Network 11
   RUNG wire#powerrail
      "Energy Saving_DB"("Start Switch" := "Start switch", "Sort IR sensor" := "Sort area IR", "System Enable Ok" := "System Run_Green Lamp", Save => "Save_Energy")
   END_RUNG
   // the same network as SCL:
   "Energy Saving_DB"("Start Switch" := "Start switch",   // "Energy Saving"
                      "Sort IR sensor" := "Sort area IR",
                      "System Enable Ok" := "System Run_Green Lamp",
                      Save => "Save_Energy");
END_REGION

REGION Network 12
   RUNG wire#powerrail
      "Alarm_DB"()
   END_RUNG
   // the same network as SCL:
   "Alarm_DB"();   // "Alarm"
END_REGION
END_ORGANIZATION_BLOCK

ORGANIZATION_BLOCK "Cyclic interrupt"   // OB30, LAD, CyclicInterrupt
TITLE = PID Controller
{ S7_Optimized_Access := 'TRUE' }
VERSION : 0.1
   VAR_INPUT
      Initial_Call : Bool;   // Initial call of this OB
      Event_Count : Int;   // Events discarded
   END_VAR
BEGIN

REGION Network 1: PID Control for oven temperature
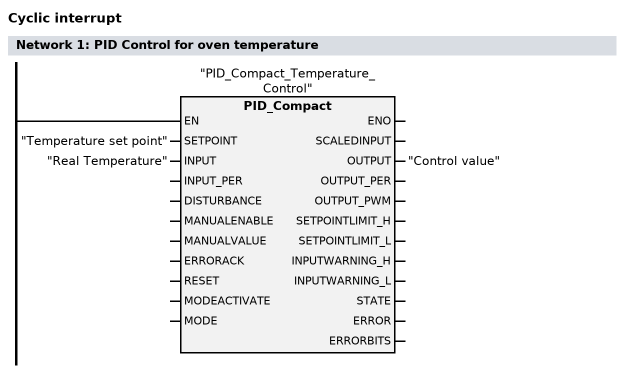
   "PID_Compact_Temperature_Control"(Setpoint := "Temperature set point",   // PID_Compact
                           Input := "Real Temperature",
                           Output => "Control value");
END_REGION
END_ORGANIZATION_BLOCK

(* ===== HMI "HMI_RT_1" =====
system functions are stored by id; their names below are inferred from use
connection "HMI_Connection_1": ETHERNET, S7_1500_OMS

HMI tags "Default tag table"
   "Counter value" : Int = PLC "Counter value" AT %MW0, 100 ms
   "Sort Solenoid Sensor" : Bool = PLC "Sort Solenoid Sensor" AT %I0.6, 100 ms
   "Ring Queue counter Full" : Bool = PLC "Ring Queue counter Full" AT %M4.0, 100 ms
   "Counter Reset" : Bool = PLC "Counter Reset" AT %M4.4, 100 ms
   "Stop switch" : Bool = PLC "Stop switch" AT %I0.3, 100 ms
   "HMI_Start" : Bool = PLC HMI_Start AT %M4.1, 100 ms
   "HMI_Stop" : Bool = PLC HMI_Stop AT %M4.2, 100 ms
   "Sort Area Inductive" : Bool = PLC "Sort Area Inductive" AT %I0.5, 100 ms
   "Sort area IR" : Bool = PLC "Sort area IR" AT %I0.4, 100 ms
   "Chain Conveyor" : Bool = PLC "Chain Conveyor" AT %Q0.0, 100 ms
   "Emergency stop" : Bool = PLC "Emergency stop" AT %I1.0, 100 ms
   "Sysyem Stop_Red Lamp" : Bool = PLC "Sysyem Stop_Red Lamp" AT %Q3.2, 100 ms
   "Panel Emergency Stop" : Bool = PLC "Panel Emergency Stop" AT %I2.7, 100 ms
   "System Run_Green Lamp" : Bool = PLC "System Run_Green Lamp" AT %Q3.0, 100 ms
   "Belt Conveyor Direction" : Bool = PLC "Belt Conveyor Direction" AT %Q0.4, 100 ms
   "Reject Solenoid Sensor" : Bool = PLC "Reject Solenoid Sensor" AT %I1.5, 100 ms
   "HMI_Emergency_Stop" : Bool = PLC HMI_Emergency_Stop AT %M5.0, 100 ms
   "Assembly Area Capacitor" : Bool = PLC "Assembly Area Capacitor" AT %I1.2, 100 ms
   "Assembly Area Inductive" : Bool = PLC "Assembly Area Inductive" AT %I1.3, 100 ms
   "Assembly Area Through Beam" : Bool = PLC "Assembly Area Through Beam" AT %I1.1, 100 ms
   "Assembly Chute IR" : Bool = PLC "Assembly Chute IR" AT %I0.7, 100 ms
   "Rotary Solenoid" : Bool = PLC "Rotary Solenoid" AT %Q0.3, 100 ms
   "Start switch" : Bool = PLC "Start switch" AT %I0.2, 100 ms
   "Reject Area IR" : Bool = PLC "Reject Area IR" AT %I1.4, 100 ms
   "Reject Solenoid" : Bool = PLC "Reject Solenoid" AT %Q0.2, 100 ms
   "Sort Solenoid" : Bool = PLC "Sort Solenoid" AT %Q0.1, 100 ms
   "Peg Counter Value" : Int = PLC "Peg Counter Value" AT %MW6, 100 ms
   "Ring Counter Value" : Int = PLC "Ring Counter Value" AT %MW2, 100 ms
   "Assembly Counter Value" : Int = PLC "Assembly Counter Value" AT %MW8, 100 ms
   "Connected" : Bool = PLC Connection_Successful AT %M5.1, 100 ms
      on ChangeValue: function_efd93a16("Connect", 0, 0, 1, 1, 1); ResetBit("Connected")
   "Disconnected" : Bool = PLC Connection_Disconnected AT %M5.2, 100 ms
      on ChangeValue: function_efd93a16("Disconnect", 0, 0, 1, 1, 1); ResetBit("Disconnected")
   "Assembly Done" : Bool = PLC HMI_AssemDone AT %M5.3, 100 ms
      on ChangeValue: function_efd93a16("Assembly Complete", 0, 0, 1, -1, 1); ResetBit("Assembly Done")
   "Real Temperature" : Real = PLC "Real Temperature" AT %MD300, 100 ms
   "ON/OFF Temperature Set Point" : Real = PLC "ON/OFF Temperature set point" AT %MD20, 100 ms
   "Temperature set point" : Real = PLC "Temperature set point" AT %MD24, 100 ms
   "Control Value" : Int = PLC "Control value" AT %MW13, 100 ms
   "Alarm_Tag" : Int = PLC Alarm_Tag AT %MW20, 100 ms
   "HMI_Reset" : Bool = PLC HMIReset AT %M6.0, 100 ms
      on ChangeValue: function_efd93a16("Assembly Complete", 0, 0, -1, -1, 1); ResetBit("HMI_Reset")

discrete alarms
   1: 'EMERGENCY STOP', class Errors, trigger "Alarm_Tag" bit 8
   2: 'PANEL EMERGENCY STOP', class Errors, trigger "Alarm_Tag" bit 9
   3: 'SORT SOLENOID ERROR', class Errors, trigger "Alarm_Tag" bit 10
   4: 'REJECT SOLENOID ERROR', class Errors, trigger "Alarm_Tag" bit 11
   5: 'Chute at maximum capacity', class Errors, trigger "Alarm_Tag" bit 12

Template "Template_1" 800x480
   Button "Exit" at 720,420 size 78x58; TextOff 'Exit'; PictureOff "ExitRuntime_TP700_Comfort_TR"; PictureOn "ExitRuntime_TP700_Comfort_TR"
      on Release: StopRuntime(0)
   Button "Template_Button" at 640,420 size 78x58; TextOff 'Text'
   Button "Template_Button_1" at 560,420 size 78x58; TextOff 'Text'
   Button "Template_Button_2" at 480,420 size 78x58; TextOff 'Text'
   Button "Template_Button_3" at 400,420 size 78x58; TextOff 'Text'
   Button "Template_Button_4" at 321,420 size 78x58; TextOff 'Text'
   Button "Template_Button_5" at 241,420 size 78x58; TextOff 'Text'
   Button "Template_Button_6" at 161,420 size 78x58; TextOff 'Text'
   Button "Alarms" at 81,420 size 78x58; TextOff 'Alarms'; PictureOff "AlarmDisplay_TP700_Comfort_TR"; PictureOn "AlarmDisplay_TP700_Comfort_TR"
      on Release: function_ef3f5d25("Alarm window_Unacknowledged", -1)
   Button "Start screen" at 1,420 size 78x58; TextOff 'Start screen'; PictureOff "NavigateHome_TP700_Comfort_TR"; PictureOn "NavigateHome_TP700_Comfort_TR"
      on Release: ActivateScreen("Sorting Station Overview", 0)

screen "Sorting Station Overview" 800x480, template "Template_1"
   Button "HmiScreenItemData_5" at 0,218 size 159x47; TextOff 'JD - Humanoid'; PictureOff "Navigates to JD - Humanoid for TP700 Comfort 15.1.0.0"; PictureOn "Navigates to JD - Humanoid for TP700 Comfort 15.1.0.0"
      on Release: ActivateScreen("JD - Humanoid", 0)
   TextField "HmiScreenItemData_6" at 80,196 size 640x25; Text 'Text'
   Button "HmiScreenItemData" at 0,10 size 159x47; TextOff 'System Control'; PictureOff "Navigates to System Control for TP700 Comfort 15.1.0.0"; PictureOn "Navigates to System Control for TP700 Comfort 15.1.0.0"
      on Release: ActivateScreen("System Control", 0)
   Button "HmiScreenItemData_1" at 0,81 size 159x47; TextOff 'Inputs/Outputs'; PictureOff "Navigates to Inputs/Outputs for TP700 Comfort 15.1.0.0"; PictureOn "Navigates to Inputs/Outputs for TP700 Comfort 15.1.0.0"
      on Release: ActivateScreen("Inputs/Outputs", 0)
   Button "HmiScreenItemData_2" at 0,149 size 159x47; TextOff 'Temperature Control'; PictureOff "Navigates to Temperature Control for TP700 Comfort 15.1.0.0"; PictureOn "Navigates to Temperature Control for TP700 Comfort 15.1.0.0"
      on Release: ActivateScreen("Temperature Control", 0)
   Button "HmiScreenItemData_7" at 0,364 size 158x47; TextOff 'System screens'; PictureOff "Navigates to System screens for TP700 Comfort 15.1.0.0"; PictureOn "Navigates to System screens for TP700 Comfort 15.1.0.0"
      on Release: ActivateScreen("System screens", 0)
   GraphicView "Graphic view_1" at 165,0 size 635x416; Picture "bytronic_jd"
   Button "HmiScreenItemData_8" at 0,291 size 159x47; TextOn 'PID Control'; TextOff 'PID Control'; PictureOff "Navigates to System screens for TP700 Comfort 15.1.0.0"; PictureOn "Navigates to System Control for TP700 Comfort 15.1.0.0"
      on Release: ActivateScreen("PID Control", 0)

screen "System Control" 800x480, template "Template_1"
   GraphicView "Graphic view_1" at 0,0 size 799x479; Picture "bytronic_2"
   Button "Button_2" at 166,389 size 36x36; TextOff 'Text'; PictureOn "Pushbutton_Round_R_On_256c"; PictureOff "Pushbutton_Round_R_Off_256c"
      on Press: function_b14e0dd5("HMI_Stop", 0)
   Button "Button_3" at 205,389 size 34x36; TextOff 'Text'; PictureOn "Pushbutton_Round_G_On_256c"; PictureOff "Pushbutton_Round_G_Off_256c"
      on Press: function_b14e0dd5("HMI_Start", 0)
   Button "Button_1" at 295,389 size 34x37; TextOff 'Text'; PictureOn "Pushbutton_Round_R_On_256c"; PictureOff "Pushbutton_Round_R_Off_256c"
      on Press: function_b14e0dd5("Counter Reset", 0)
   IOField "I/O field_1" at 50,306 size 43x27; FormatPattern s9
      ProcessValue <- "Counter value"
   Circle "Circle_2" at 99,306 size 26x26
      Appearance <- "Ring Queue counter Full"
   TextField "Text field_1" at 45,286 size 115x20; Text 'Counter Value'
   Circle "Circle_1" at 260,40 size 11x11
      Appearance <- "Sort Solenoid Sensor"
   Button "Back" at 1,1 size 159x47; TextOn 'Back'; TextOff 'Back'
      on Release: ActivateScreen("Sorting Station Overview", 0)
   Circle "Circle_3" at 260,111 size 14x14
      Appearance <- "Sort Area Inductive"
   Rectangle "Rectangle_1" at 245,102 size 4x23
      Appearance <- "Sort area IR"
   Ellipse "Ellipse_1" at 166,135 size 11x11
      Appearance <- "Chain Conveyor"
   Circle "Circle_4" at 416,366 size 23x23
      Appearance <- "Sysyem Stop_Red Lamp"
   Circle "Circle_5" at 417,389 size 22x22
      Appearance <- "Emergency stop"
   Circle "Circle_6" at 417,411 size 23x23
      Appearance <- "System Run_Green Lamp"
   Circle "Circle_7" at 493,332 size 10x10
      Appearance <- "Reject Solenoid Sensor"
   Circle "Circle_8" at 510,301 size 11x11
      Appearance <- "Belt Conveyor Direction"
   Circle "Circle_9" at 323,261 size 14x14
      Appearance <- "Assembly Area Inductive"
   Ellipse "Ellipse_2" at 319,214 size 23x12
      Appearance <- "Assembly Area Capacitor"
   Circle "Circle_10" at 351,242 size 12x12
      Appearance <- "Assembly Area Through Beam"
   Rectangle "Rectangle_2" at 260,286 size 15x6
      Appearance <- "Assembly Chute IR"
   Circle "Circle_11" at 264,252 size 7x7
      Appearance <- "Rotary Solenoid"
   GraphicView "Graphic view_2" at 363,12 size 54x55; Picture "peg"
   GraphicView "Graphic view_3" at 432,12 size 57x54; Picture "Ring"
   GraphicView "Graphic view_4" at 507,12 size 59x52; Picture "Assembly Done"
   IOField "I/O field_2" at 368,61 size 43x27; FormatPattern s9
      ProcessValue <- "Peg Counter Value"
   IOField "I/O field_3" at 440,62 size 43x27; FormatPattern s9
      ProcessValue <- "Ring Counter Value"
   IOField "I/O field_4" at 515,61 size 43x27; FormatPattern s9
      ProcessValue <- "Assembly Counter Value"
   Button "Button_4" at 59,379 size 51x51; TextOff 'Text'; PictureOn "PilotLight_Round_R_On_256c"; PictureOff "Pushbutton_Round_R_Off_256c"
      on Press: function_b14e0dd5("HMI_Emergency_Stop", 0)

screen "Inputs/Outputs" 800x480, template "Template_1"
   Button "Back" at 1,1 size 159x47; TextOff 'Back'
      on Release: ActivateScreen("Sorting Station Overview", 0)
   TextField "Text field_1" at 15,60 size 134x23; Text 'Counter Value'
   TextField "Text field_2" at 289,56 size 63x23; Text 'Inputs'
   TextField "Text field_3" at 638,56 size 76x23; Text 'Outputs'
   Bar "Bar_1" at 34,124 size 80x230; MinimumValue 0; MaximumValue 6
      ProcessValue <- "Counter value"
   Button "Button_1" at 158,84 size 108x32; TextOff 'Start Switch'
      Appearance <- "Start switch"
   Button "Button_2" at 349,83 size 144x32; TextOff 'Stop Switch'
      Appearance <- "Stop switch"
   Button "Button_3" at 158,111 size 118x32; TextOff 'Sort Area IR'
      Appearance <- "Sort area IR"
   Button "Button_4" at 158,141 size 172x32; TextOff 'Sort Area Inductive'
      Appearance <- "Sort Area Inductive"
   Button "Button_5" at 158,171 size 181x32; TextOff 'Sort Solenoid Sensor'
      Appearance <- "Sort Solenoid Sensor"
   Button "Button_7" at 159,231 size 214x32; TextOff 'Assembly Area Inductive'
      Appearance <- "Assembly Area Inductive"
   Button "Button_8" at 159,286 size 253x32; TextOff 'Assembly Area Through Beam'
      Appearance <- "Assembly Area Through Beam"
   Button "Button_9" at 160,316 size 255x32; TextOff 'Reject Area IR'
      Appearance <- "Reject Area IR"
   Button "Button_10" at 160,345 size 255x32; TextOff 'Reject Solenoid'
      Appearance <- "Reject Solenoid"
   Button "Button_11" at 349,111 size 194x32; TextOff 'Panel Emergency Stop'
      Appearance <- "Panel Emergency Stop"
   Button "Button_12" at 558,83 size 211x32; TextOff 'Chain Conveyor'
      Appearance <- "Chain Conveyor"
   Button "Button_13" at 559,115 size 211x32; TextOff 'Sort Solenoid'
      Appearance <- "Sort Solenoid"
   Button "Button_14" at 559,143 size 211x32; TextOff 'Reject Solenoid'
      Appearance <- "Reject Solenoid"
   Button "Button_15" at 560,174 size 210x32; TextOff 'Rotary Solenoid'
      Appearance <- "Rotary Solenoid"
   Button "Button_16" at 560,205 size 210x32; TextOff 'Belt Conveyor'
      Appearance <- "Belt Conveyor Direction"
   Button "Button_17" at 560,235 size 210x32; TextOff 'System Run Green'
      Appearance <- "System Run_Green Lamp"
   Button "Button_18" at 560,265 size 211x32; TextOff 'System Stop Red'
      Appearance <- "Sysyem Stop_Red Lamp"
   Button "Button_19" at 158,199 size 189x32; TextOff 'Assembly Chute IR'
      Appearance <- "Assembly Chute IR"
   Button "Button_20" at 349,142 size 193x32; TextOff 'Emergency Stop'
      Appearance <- "Emergency stop"
   Button "Button_6" at 159,259 size 219x32; TextOff 'Assembly Area Capacitive'
      Appearance <- "Assembly Area Capacitor"

screen "Temperature Control" 800x480, template "Template_1"
   TextField "HmiScreenItemData" at 80,196 size 640x25; Text 'Temperature Control'
   Button "Back" at 1,1 size 159x47; TextOff 'Back'
      on Release: ActivateScreen("Sorting Station Overview", 0)

screen "JD - Humanoid" 800x480, template "Template_1"
   GraphicView "Graphic view_1" at 0,1 size 800x478; Picture "jd"
   Button "Back" at 1,1 size 159x47; TextOff 'Back'
      on Release: ActivateScreen("Sorting Station Overview", 0)

screen "System screens" 800x480, template "Template_1"
   Button "Back" at 1,1 size 159x47; TextOff 'Back'
      on Release: ActivateScreen("Sorting Station Overview", 0)
   Button "HmiScreenItemData" at 36,95 size 159x47; TextOff 'SIMATIC PLC system diagnos...'; PictureOff "Navigates to SIMATIC PLC system diagnostics for TP700 Comfort 15.1.0.0"; PictureOn "Navigates to SIMATIC PLC system diagnostics for TP700 Comfort 15.1.0.0"
      on Release: ActivateScreen("SIMATIC PLC system diagnostics", 0)

screen "SIMATIC PLC system diagnostics" 800x480, template "Template_1"
   SysDiagControl "HmiScreenItemData" at 1,49 size 796x364
   Button "Back" at 1,1 size 159x47; TextOff 'Back'
      on Release: ActivateScreen("System screens", 0)

PopupScreen "Connect" 240x240
   TextField "Text field_1" at 25,156 size 215x23; Text 'Connected Successfully'
   Button "Button_1" at 143,206 size 96x32; TextOff 'Exit'
      on Press: function_efd93a16("Connect", 0, 0, 0, -1, 1)
   GraphicView "Graphic view_1" at 46,27 size 144x101; Picture "JD_Conn_1"

PopupScreen "Assembly Complete" 240x240
   TextField "Text field_1" at 32,111 size 193x23; Text 'Assembly Completed'
   Button "Button_1" at 142,208 size 96x32; TextOff 'Exit'
      on Press: function_efd93a16("Assembly Complete", 0, 0, 0, -1, 1)
   GraphicView "Graphic view_1" at 68,24 size 96x82; Picture "Assembly Done"

PopupScreen "Disconnect" 240x240
   TextField "Text field_1" at 65,159 size 125x23; Text 'Disconnected'
   Button "Button_1" at 144,208 size 96x32; TextOff 'Exit'
      on Press: function_efd93a16("Disconnect", 0, 0, 0, -1, 1)
   GraphicView "Graphic view_1" at 38,25 size 154x113; Picture "JD_Discon"

screen "PID Control" 800x480
   Button "Back" at 0,433 size 159x47; TextOn 'Back'; TextOff 'Back'
      on Release: ActivateScreen("Sorting Station Overview", 0)
   TrendView "Trend view_1" at 0,0 size 800x433
   IOField "I/O field_1" at 697,433 size 102x46; FormatPattern s99
      ProcessValue <- "Temperature set point"
   TextField "Text field_1" at 492,445 size 226x23; Text 'Temperature Set Point:'
*)